FUNCTION_BLOCK PAMIntermediatebin EXTENDS PAProcessModule
VAR_INPUT
END_VAR
VAR_OUTPUT
END_VAR
VAR
	_PAPointMatIn1 : PAPoint(THIS^);
	_PAPointMatOut1 : PAPoint(THIS^);
END_VAR

METHOD FB_init : BOOL
VAR_INPUT
	bInitRetains : BOOL; // if TRUE, the retain variables are initialized (warm start / cold start)
	bInCopyCode : BOOL;  // if TRUE, the instance afterwards gets moved into the copy code (online change)
	parent : IACComponent;
END_VAR
AddPoint(_PAPointMatIn1);
AddPoint(_PAPointMatOut1);
END_METHOD

PROPERTY PUBLIC PAPointMatIn1 : IACPoint
GET
PAPointMatIn1 := _PAPointMatIn1;
END_GET
END_PROPERTY

PROPERTY PUBLIC PAPointMatOut1 : IACPoint
GET
PAPointMatOut1 := _PAPointMatOut1;
END_GET
END_PROPERTY

END_FUNCTION_BLOCK

(* stored: Version 1.1.0.1, ProductVersion 3.1.4020.12
   POU PAMIntermediatebin: Id {cf215125-1076-46ce-a17c-b50191dc88e0}, SpecialFunc None
   Method FB_init: Id {85f1e6ef-c51e-497d-b4e0-0e7c851d4312}
   Property PAPointMatIn1: Id {277af98b-5a21-49a3-a1f6-df0ab5c8b96d}
   Get Get: Id {768eb1d0-63ef-4fa5-9fd5-43b4f748751f}
   Property PAPointMatOut1: Id {43712bb8-c496-4a7e-ad03-76d6e5225338}
   Get Get: Id {e18fffe4-005b-49c6-9d9d-4036802b1bf7} *)
